{attribute 'linkalways'} 
{attribute 'no_explicit_call' := 'This FB is a CLASS and must be accessed using methods or properties'}
{attribute 'enable_dynamic_creation'}
FUNCTION_BLOCK TaskCyclicEvent EXTENDS Event IMPLEMENTS I_TaskCyclicEvent
VAR
	parent : I_Task;
END_VAR

METHOD FB_init : BOOL
VAR_INPUT
	bInitRetains : BOOL; // if TRUE, the retain variables are initialized (warm start / cold start)
	bInCopyCode : BOOL;  // if TRUE, the instance afterwards gets moved into the copy code (online change)
	Parent : I_Task;
END_VAR
this^.parent := Parent;
END_METHOD

PROPERTY Info : PlcTaskSystemInfo
GET
Info := parent.Info;
END_GET
END_PROPERTY

METHOD PUBLIC Notify
VAR_INPUT
END_VAR
NotifySubscribers();
END_METHOD

END_FUNCTION_BLOCK

(* stored: Version 1.1.0.1, ProductVersion 3.1.4024.12
   POU TaskCyclicEvent: Id {686a8a4b-99a9-065c-0368-7459b592e8e9}, SpecialFunc None
   Method FB_init: Id {a48499b0-f0fa-06a5-1784-c4068ff83a2d}
   Property Info: Id {d5dcf704-e168-0658-333f-e30fa58fb990}
   Get Get: Id {f81117be-3638-04da-0db8-2a28defa47de}
   Method Notify: Id {ec0f4aa7-237c-03d6-0a35-cb2658141257} *)
